(* CODESYS project myRepo001

Project tree, tasks and I/O mapping:
  Device : CODESYS Control for PFC200 SL, 3S - Smart Software Solutions GmbH, version 4.3.0.0
    application Application
      libraries: Standard, 3.5.18.0 (System)
      task MainTask (cyclic, interval t#20ms, priority 1) calls PLC_PRG
      program PLC_PRG [ST]
    Pfc200Bus : Wago PFC200 internal bus, 3S - Smart Software Solutions GmbH, version 4.3.0.0
*)

// Device/Application/PLC_PRG
PROGRAM PLC_PRG
VAR
	a: INT;
END_VAR

a:=a+1;

END_PROGRAM
